{attribute 'GeneratedUsingTerminal: EL5101-0000-1020'}
{attribute addProperty BoxType "EL5101-0000-1020"}
{attribute addProperty Id "StatusAT %I*Status_6D6CFE2016Counter_valueAT %I*UINT2Latch_valueAT %I*UINT2"}
{attribute addProperty CRC "1866614104"}
{attribute addProperty Size "20"}
TYPE ENC_Status_compact_6F424558 :
STRUCT
	{attribute addProperty Name "Status"}
	Status AT %I* : Status_6D6CFE20;
	{attribute addProperty Name "Counter_value"}
	Counter_value AT %I* : UINT;
	{attribute addProperty Name "Latch_value"}
	Latch_value AT %I* : UINT;
END_STRUCT
END_TYPE

(* stored: Version 1.2.0.0, ProductVersion 3.1.4024.9
   DUT ENC_Status_compact_6F424558: Id {7928eb56-cd21-4d95-b16e-2e2662e04386} *)
